FUNCTION_BLOCK SPLIT_SIGNED_LINT (* Teilt einen LINT-Wert in 2 einseitige Betragswerte auf: NEG_MAG = MAX(0,-Y), POS_MAG = MAX(0,Y). Sonderfall Y=LINT#-9223372036854775808 (LINT-Minimum): -Y wuerde ueberlaufen (Zweierkomplement, |MIN| > MAX) - in diesem Fall wird NEG_MAG auf LINT#9223372036854775807 (LINT-Maximum) begrenzt (Regelungstechnik: Saettigung statt Ueberlauf/Vorzeichenwechsel). Feuert CNF bei jedem REQ, unabhaengig von Wertaenderung - Event-Deduplizierung erfolgt aussen im Adapter-Wrapper ALI_SPLIT_SIGNED ueber je einen E_D_FF_ANY pro Seite. *)
  (* Standard: 61499-2 *)
  (* Version 1.0, 2026-09-11, Franz Höpfinger, Einfacher Value/Event-Baustein ohne Event-Dedup - wird vom Adapter-Wrapper ALI_SPLIT_SIGNED mit je einem E_D_FF_ANY pro Seite dedupliziert *)
  PACKAGE adapter::Engineering::splitting::signed;
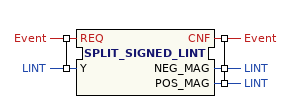
  EVENT_INPUT
    REQ WITH Y; (* Neuer Y-Wert liegt an *)
  END_EVENT
  EVENT_OUTPUT
    CNF WITH NEG_MAG, POS_MAG; (* NEG_MAG/POS_MAG berechnet *)
  END_EVENT
  VAR_INPUT
    Y : LINT; (* Eingangswert *)
  END_VAR
  VAR_OUTPUT
    NEG_MAG : LINT; (* MAX(0, -Y), bei Y=LINT#-9223372036854775808 gesaettigt auf LINT#9223372036854775807 *)
    POS_MAG : LINT; (* MAX(0, Y) *)
  END_VAR
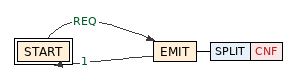
  EC_STATES
    START; (* Initial State *)
    EMIT : SPLIT -> CNF;
  END_STATES
  EC_TRANSITIONS
    START TO EMIT := REQ;
    EMIT TO START := 1;
  END_TRANSITIONS
  ALGORITHM SPLIT IN ST:
IF Y = LINT#-9223372036854775808 THEN
	NEG_MAG := LINT#9223372036854775807;
ELSE
	NEG_MAG := MAX(LINT#0,-Y);
END_IF;
POS_MAG := MAX(LINT#0,Y);
  END_ALGORITHM
END_FUNCTION_BLOCK
